// Mitsubishi GX Works2 project: Step Control   PLC: Q01U

PROGRAM conveyor
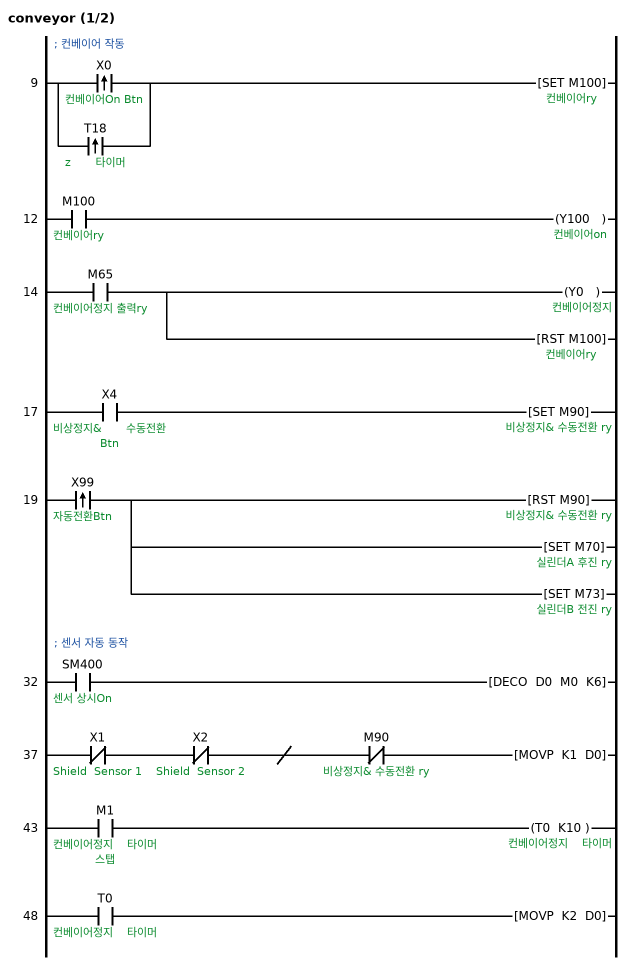
; 컨베이어 작동
9     LDP     X0  ; 컨베이어On Btn
      ORP     T18  ; z       타이머
      SET     M100  ; 컨베이어ry
12    LD      M100  ; 컨베이어ry
      OUT     Y100  ; 컨베이어on
14    LD      M65  ; 컨베이어정지 출력ry
      OUT     Y0  ; 컨베이어정지
      RST     M100  ; 컨베이어ry
17    LD      X4  ; 비상정지&       수동전환 Btn
      SET     M90  ; 비상정지& 수동전환 ry
19    LDP     X99  ; 자동전환Btn
      RST     M90  ; 비상정지& 수동전환 ry
      SET     M70  ; 실린더A 후진 ry
      SET     M73  ; 실린더B 전진 ry
; 센서 자동 동작
32    LD      SM400  ; 센서 상시On
      DECO    D0 M0 K6
37    LDI     X1  ; Shield  Sensor 1
      ANI     X2  ; Shield  Sensor 2
      INV
      ANI     M90  ; 비상정지& 수동전환 ry
      MOVP    K1 D0
43    LD      M1  ; 컨베이어정지    타이머  스탭
      OUT     T0 K10  ; 컨베이어정지    타이머
48    LD      T0  ; 컨베이어정지    타이머
      MOVP    K2 D0
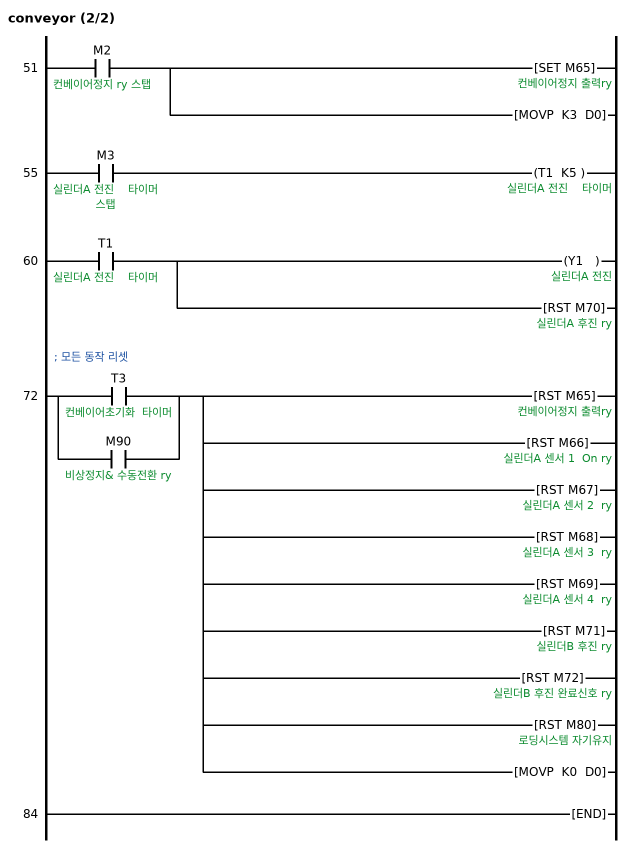
51    LD      M2  ; 컨베이어정지 ry 스탭
      SET     M65  ; 컨베이어정지 출력ry
      MOVP    K3 D0
55    LD      M3  ; 실린더A 전진    타이머  스탭
      OUT     T1 K5  ; 실린더A 전진    타이머
60    LD      T1  ; 실린더A 전진    타이머
      OUT     Y1  ; 실린더A 전진
      RST     M70  ; 실린더A 후진 ry
; 모든 동작 리셋
72    LD      T3  ; 컨베이어초기화  타이머
      OR      M90  ; 비상정지& 수동전환 ry
      RST     M65  ; 컨베이어정지 출력ry
      RST     M66  ; 실린더A 센서 1  On ry
      RST     M67  ; 실린더A 센서 2  ry
      RST     M68  ; 실린더A 센서 3  ry
      RST     M69  ; 실린더A 센서 4  ry
      RST     M71  ; 실린더B 후진 ry
      RST     M72  ; 실린더B 후진 완료신호 ry
      RST     M80  ; 로딩시스템 자기유지
      MOVP    K0 D0
84    END
END_PROGRAM

PROGRAM cylinder
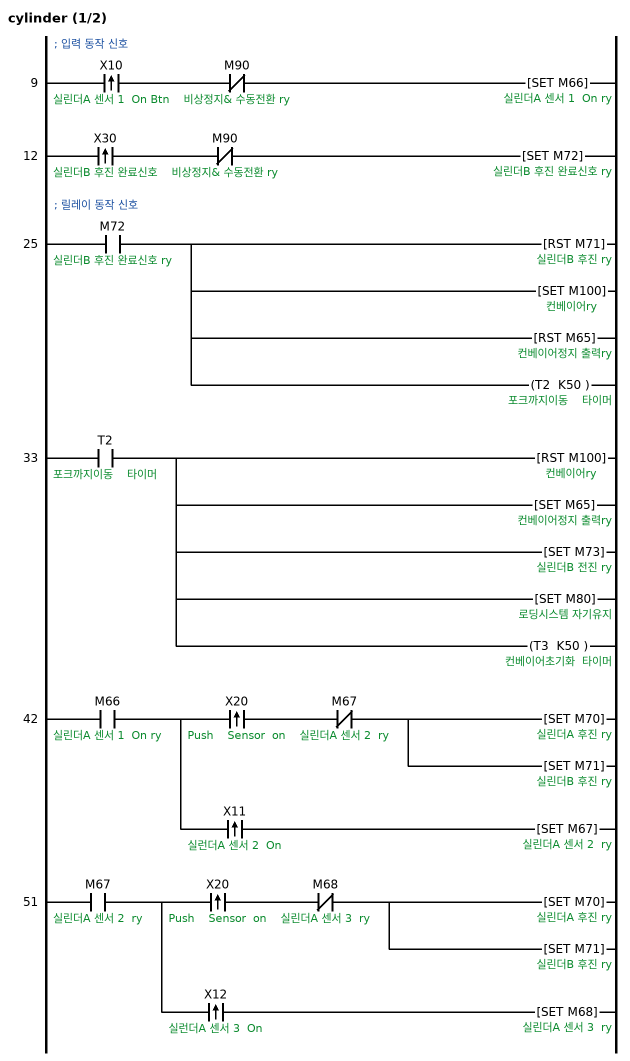
; 입력 동작 신호
9     LDP     X10  ; 실린더A 센서 1  On Btn
      ANI     M90  ; 비상정지& 수동전환 ry
      SET     M66  ; 실린더A 센서 1  On ry
12    LDP     X30  ; 실린더B 후진 완료신호
      ANI     M90  ; 비상정지& 수동전환 ry
      SET     M72  ; 실린더B 후진 완료신호 ry
; 릴레이 동작 신호
25    LD      M72  ; 실린더B 후진 완료신호 ry
      RST     M71  ; 실린더B 후진 ry
      SET     M100  ; 컨베이어ry
      RST     M65  ; 컨베이어정지 출력ry
      OUT     T2 K50  ; 포크까지이동    타이머
33    LD      T2  ; 포크까지이동    타이머
      RST     M100  ; 컨베이어ry
      SET     M65  ; 컨베이어정지 출력ry
      SET     M73  ; 실린더B 전진 ry
      SET     M80  ; 로딩시스템 자기유지
      OUT     T3 K50  ; 컨베이어초기화  타이머
42    LD      M66  ; 실린더A 센서 1  On ry
      MPS
      ANDP    X20  ; Push    Sensor  on
      ANI     M67  ; 실린더A 센서 2  ry
      SET     M70  ; 실린더A 후진 ry
      SET     M71  ; 실린더B 후진 ry
      MPP
      ANDP    X11  ; 실런더A 센서 2  On
      SET     M67  ; 실린더A 센서 2  ry
51    LD      M67  ; 실린더A 센서 2  ry
      MPS
      ANDP    X20  ; Push    Sensor  on
      ANI     M68  ; 실린더A 센서 3  ry
      SET     M70  ; 실린더A 후진 ry
      SET     M71  ; 실린더B 후진 ry
      MPP
      ANDP    X12  ; 실런더A 센서 3  On
      SET     M68  ; 실린더A 센서 3  ry
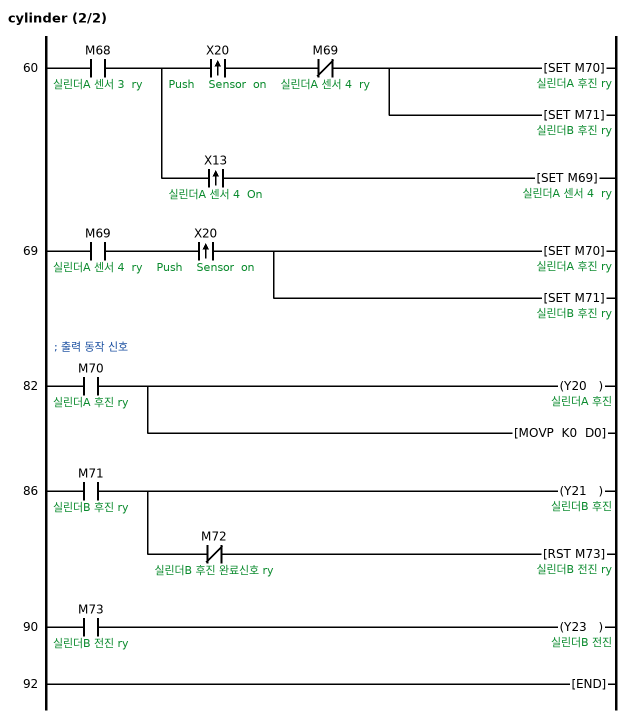
60    LD      M68  ; 실린더A 센서 3  ry
      MPS
      ANDP    X20  ; Push    Sensor  on
      ANI     M69  ; 실린더A 센서 4  ry
      SET     M70  ; 실린더A 후진 ry
      SET     M71  ; 실린더B 후진 ry
      MPP
      ANDP    X13  ; 실린더A 센서 4  On
      SET     M69  ; 실린더A 센서 4  ry
69    LD      M69  ; 실린더A 센서 4  ry
      ANDP    X20  ; Push    Sensor  on
      SET     M70  ; 실린더A 후진 ry
      SET     M71  ; 실린더B 후진 ry
; 출력 동작 신호
82    LD      M70  ; 실린더A 후진 ry
      OUT     Y20  ; 실린더A 후진
      MOVP    K0 D0
86    LD      M71  ; 실린더B 후진 ry
      OUT     Y21  ; 실린더B 후진
      ANI     M72  ; 실린더B 후진 완료신호 ry
      RST     M73  ; 실린더B 전진 ry
90    LD      M73  ; 실린더B 전진 ry
      OUT     Y23  ; 실린더B 전진
92    END
END_PROGRAM

PROGRAM manual
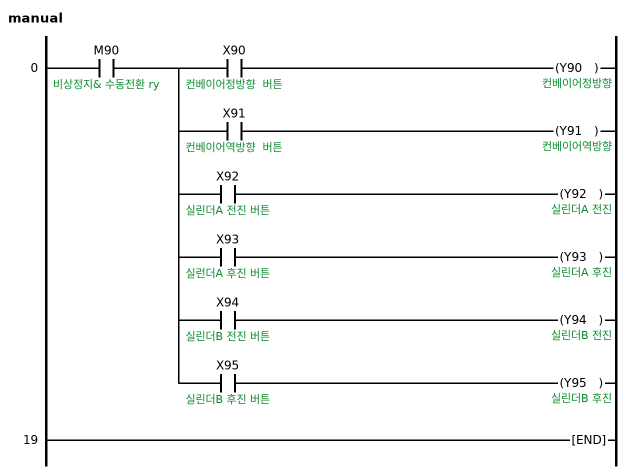
0     LD      M90  ; 비상정지& 수동전환 ry
      MPS
      AND     X90  ; 컨베이어정방향  버튼
      OUT     Y90  ; 컨베이어정방향
      MRD
      AND     X91  ; 컨베이어역방향  버튼
      OUT     Y91  ; 컨베이어역방향
      MRD
      AND     X92  ; 실린더A 전진 버튼
      OUT     Y92  ; 실린더A 전진
      MRD
      AND     X93  ; 실런더A 후진 버튼
      OUT     Y93  ; 실린더A 후진
      MRD
      AND     X94  ; 실린더B 전진 버튼
      OUT     Y94  ; 실린더B 전진
      MPP
      AND     X95  ; 실린더B 후진 버튼
      OUT     Y95  ; 실린더B 후진
19    END
END_PROGRAM

PROGRAM boxSize
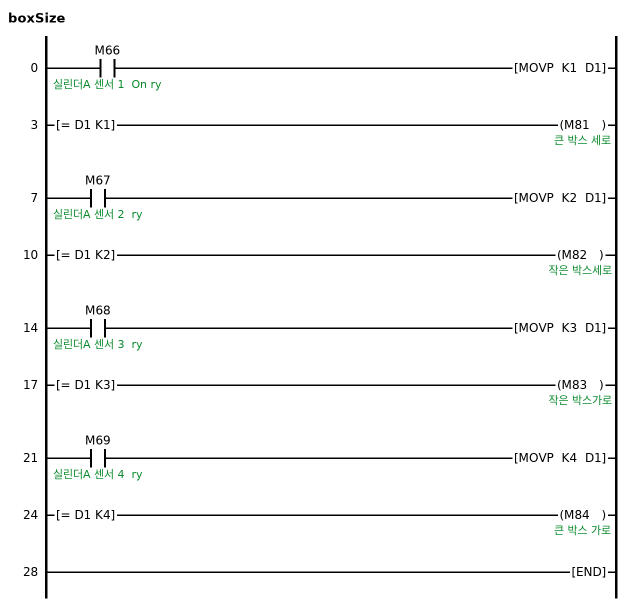
0     LD      M66  ; 실린더A 센서 1  On ry
      MOVP    K1 D1
3     LD=     D1 K1
      OUT     M81  ; 큰 박스 세로
7     LD      M67  ; 실린더A 센서 2  ry
      MOVP    K2 D1
10    LD=     D1 K2
      OUT     M82  ; 작은 박스세로
14    LD      M68  ; 실린더A 센서 3  ry
      MOVP    K3 D1
17    LD=     D1 K3
      OUT     M83  ; 작은 박스가로
21    LD      M69  ; 실린더A 센서 4  ry
      MOVP    K4 D1
24    LD=     D1 K4
      OUT     M84  ; 큰 박스 가로
28    END
END_PROGRAM

PROGRAM Box4move
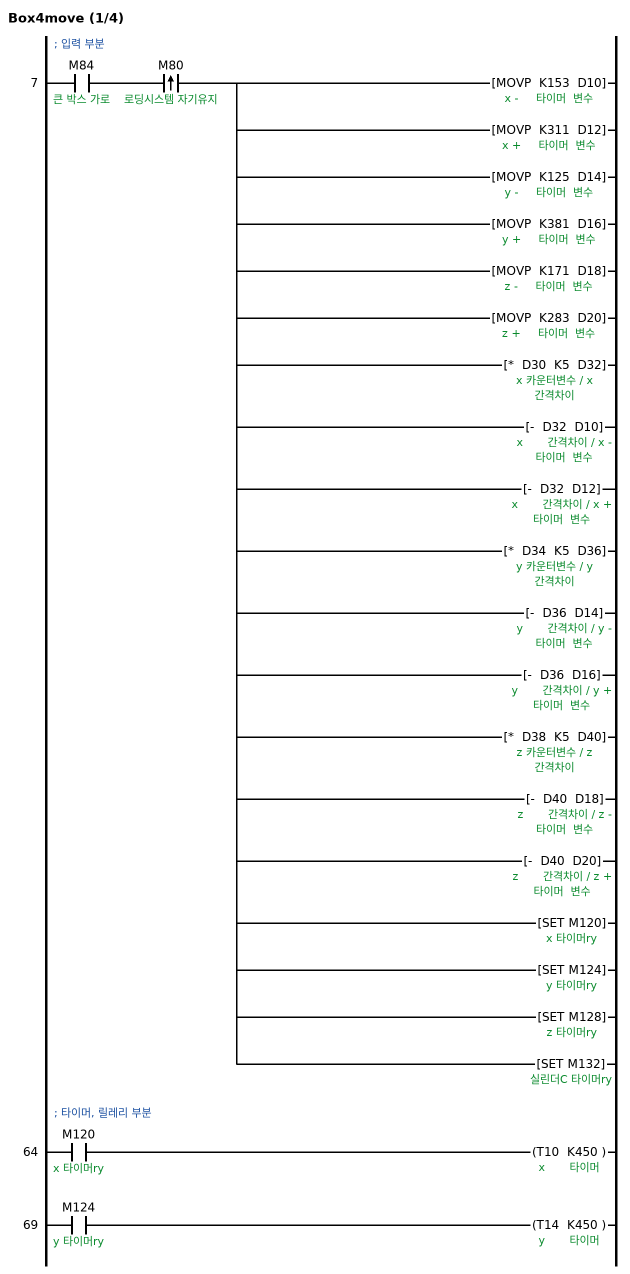
; 입력 부분
7     LD      M84  ; 큰 박스 가로
      ANDP    M80  ; 로딩시스템 자기유지
      MOVP    K153 D10  ; x -     타이머  변수
      MOVP    K311 D12  ; x +     타이머  변수
      MOVP    K125 D14  ; y -     타이머  변수
      MOVP    K381 D16  ; y +     타이머  변수
      MOVP    K171 D18  ; z -     타이머  변수
      MOVP    K283 D20  ; z +     타이머  변수
      *       D30 K5 D32  ; x 카운터변수 / x       간격차이
      -       D32 D10
      -       D32 D12
      *       D34 K5 D36  ; y 카운터변수 / y       간격차이
      -       D36 D14
      -       D36 D16
      *       D38 K5 D40  ; z 카운터변수 / z       간격차이
      -       D40 D18
      -       D40 D20
      SET     M120  ; x 타이머ry
      SET     M124  ; y 타이머ry
      SET     M128  ; z 타이머ry
      SET     M132  ; 실린더C 타이머ry
; 타이머, 릴레리 부분
64    LD      M120  ; x 타이머ry
      OUT     T10 K450  ; x       타이머
69    LD      M124  ; y 타이머ry
      OUT     T14 K450  ; y       타이머
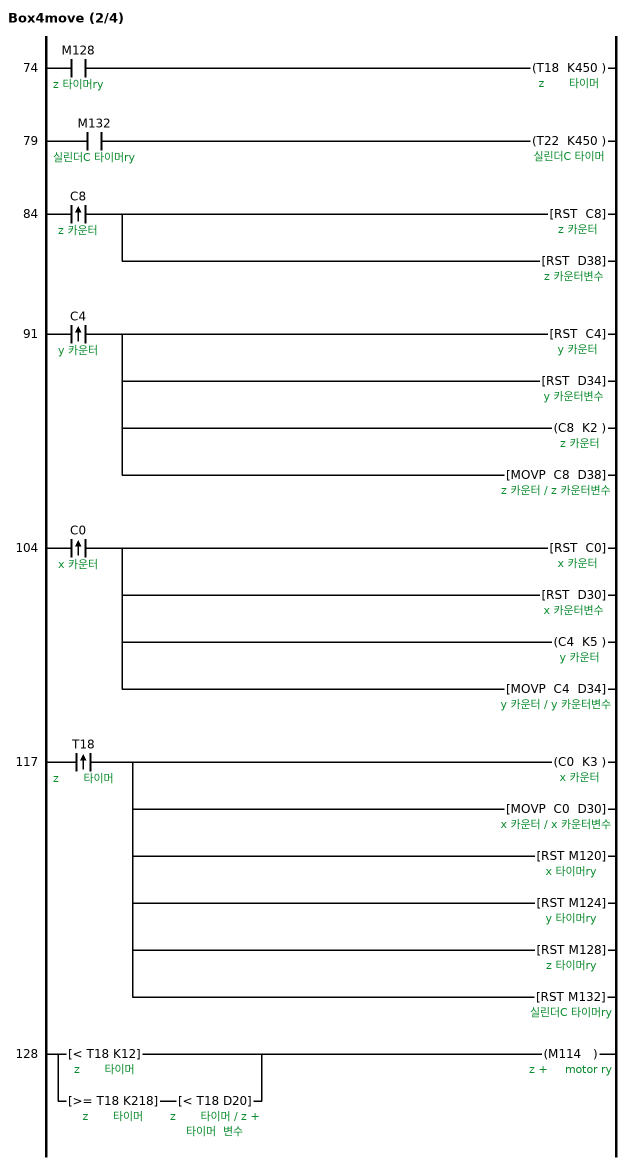
74    LD      M128  ; z 타이머ry
      OUT     T18 K450  ; z       타이머
79    LD      M132  ; 실린더C 타이머ry
      OUT     T22 K450  ; 실린더C 타이머
84    LDP     C8  ; z 카운터
      RST     C8  ; z 카운터
      RST     D38  ; z 카운터변수
91    LDP     C4  ; y 카운터
      RST     C4  ; y 카운터
      RST     D34  ; y 카운터변수
      OUT     C8 K2  ; z 카운터
      MOVP    C8 D38
104   LDP     C0  ; x 카운터
      RST     C0  ; x 카운터
      RST     D30  ; x 카운터변수
      OUT     C4 K5  ; y 카운터
      MOVP    C4 D34
117   LDP     T18  ; z       타이머
      OUT     C0 K3  ; x 카운터
      MOVP    C0 D30
      RST     M120  ; x 타이머ry
      RST     M124  ; y 타이머ry
      RST     M128  ; z 타이머ry
      RST     M132  ; 실린더C 타이머ry
128   LD<     T18 K12  ; z       타이머
      LD>=    T18 K218  ; z       타이머
      AND<    T18 D20  ; z       타이머 / z +     타이머  변수
      ORB
      OUT     M114  ; z +     motor ry
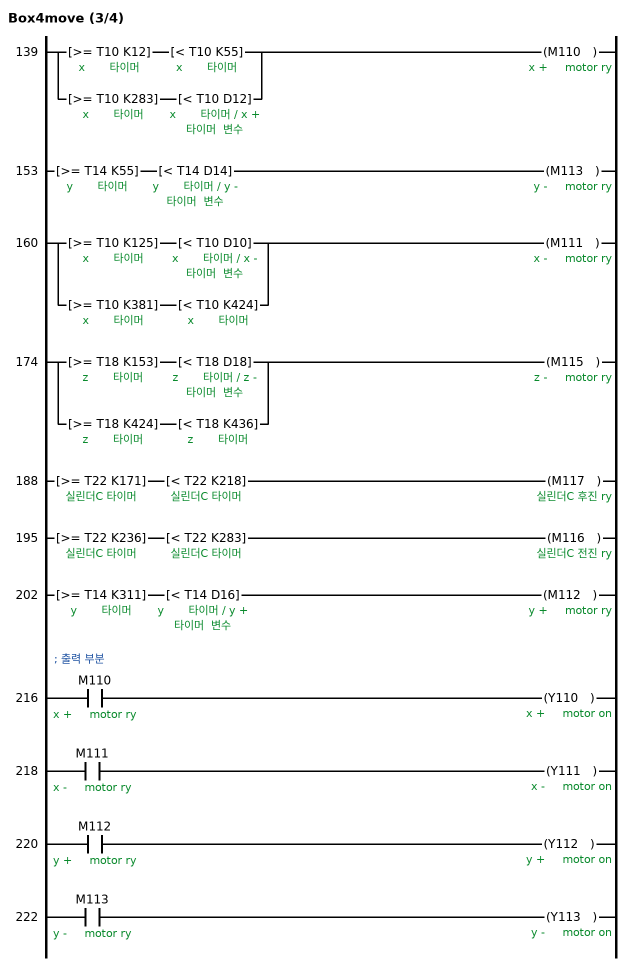
139   LD>=    T10 K12  ; x       타이머
      AND<    T10 K55  ; x       타이머
      LD>=    T10 K283  ; x       타이머
      AND<    T10 D12  ; x       타이머 / x +     타이머  변수
      ORB
      OUT     M110  ; x +     motor ry
153   LD>=    T14 K55  ; y       타이머
      AND<    T14 D14  ; y       타이머 / y -     타이머  변수
      OUT     M113  ; y -     motor ry
160   LD>=    T10 K125  ; x       타이머
      AND<    T10 D10  ; x       타이머 / x -     타이머  변수
      LD>=    T10 K381  ; x       타이머
      AND<    T10 K424  ; x       타이머
      ORB
      OUT     M111  ; x -     motor ry
174   LD>=    T18 K153  ; z       타이머
      AND<    T18 D18  ; z       타이머 / z -     타이머  변수
      LD>=    T18 K424  ; z       타이머
      AND<    T18 K436  ; z       타이머
      ORB
      OUT     M115  ; z -     motor ry
188   LD>=    T22 K171  ; 실린더C 타이머
      AND<    T22 K218  ; 실린더C 타이머
      OUT     M117  ; 실린더C 후진 ry
195   LD>=    T22 K236  ; 실린더C 타이머
      AND<    T22 K283  ; 실린더C 타이머
      OUT     M116  ; 실린더C 전진 ry
202   LD>=    T14 K311  ; y       타이머
      AND<    T14 D16  ; y       타이머 / y +     타이머  변수
      OUT     M112  ; y +     motor ry
; 출력 부분
216   LD      M110  ; x +     motor ry
      OUT     Y110  ; x +     motor on
218   LD      M111  ; x -     motor ry
      OUT     Y111  ; x -     motor on
220   LD      M112  ; y +     motor ry
      OUT     Y112  ; y +     motor on
222   LD      M113  ; y -     motor ry
      OUT     Y113  ; y -     motor on
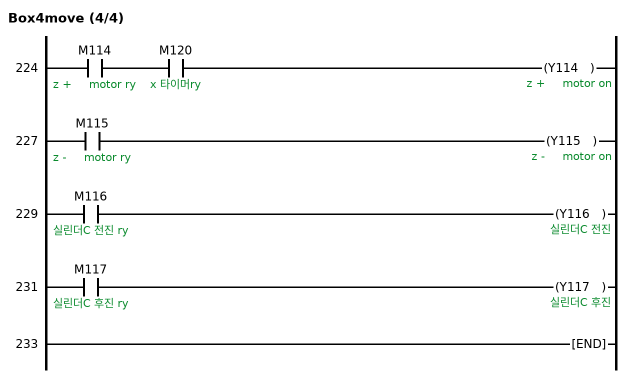
224   LD      M114  ; z +     motor ry
      AND     M120  ; x 타이머ry
      OUT     Y114  ; z +     motor on
227   LD      M115  ; z -     motor ry
      OUT     Y115  ; z -     motor on
229   LD      M116  ; 실린더C 전진 ry
      OUT     Y116  ; 실린더C 전진
231   LD      M117  ; 실린더C 후진 ry
      OUT     Y117  ; 실린더C 후진
233   END
END_PROGRAM

PROGRAM Lmanual
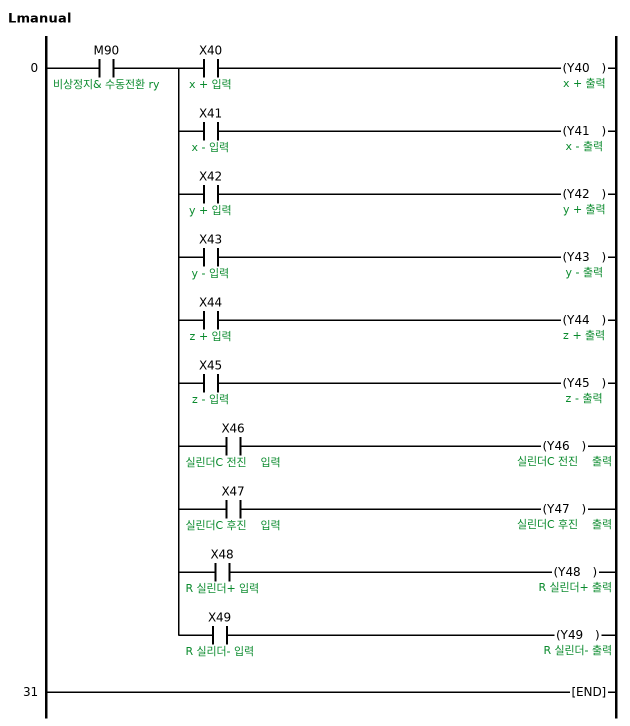
0     LD      M90  ; 비상정지& 수동전환 ry
      MPS
      AND     X40  ; x + 입력
      OUT     Y40  ; x + 출력
      MRD
      AND     X41  ; x - 입력
      OUT     Y41  ; x - 출력
      MRD
      AND     X42  ; y + 입력
      OUT     Y42  ; y + 출력
      MRD
      AND     X43  ; y - 입력
      OUT     Y43  ; y - 출력
      MRD
      AND     X44  ; z + 입력
      OUT     Y44  ; z + 출력
      MRD
      AND     X45  ; z - 입력
      OUT     Y45  ; z - 출력
      MRD
      AND     X46  ; 실린더C 전진    입력
      OUT     Y46  ; 실린더C 전진    출력
      MRD
      AND     X47  ; 실린더C 후진    입력
      OUT     Y47  ; 실린더C 후진    출력
      MRD
      AND     X48  ; R 실린더+ 입력
      OUT     Y48  ; R 실린더+ 출력
      MPP
      AND     X49  ; R 실리더- 입력
      OUT     Y49  ; R 실린더- 출력
31    END
END_PROGRAM

PROGRAM Box1move
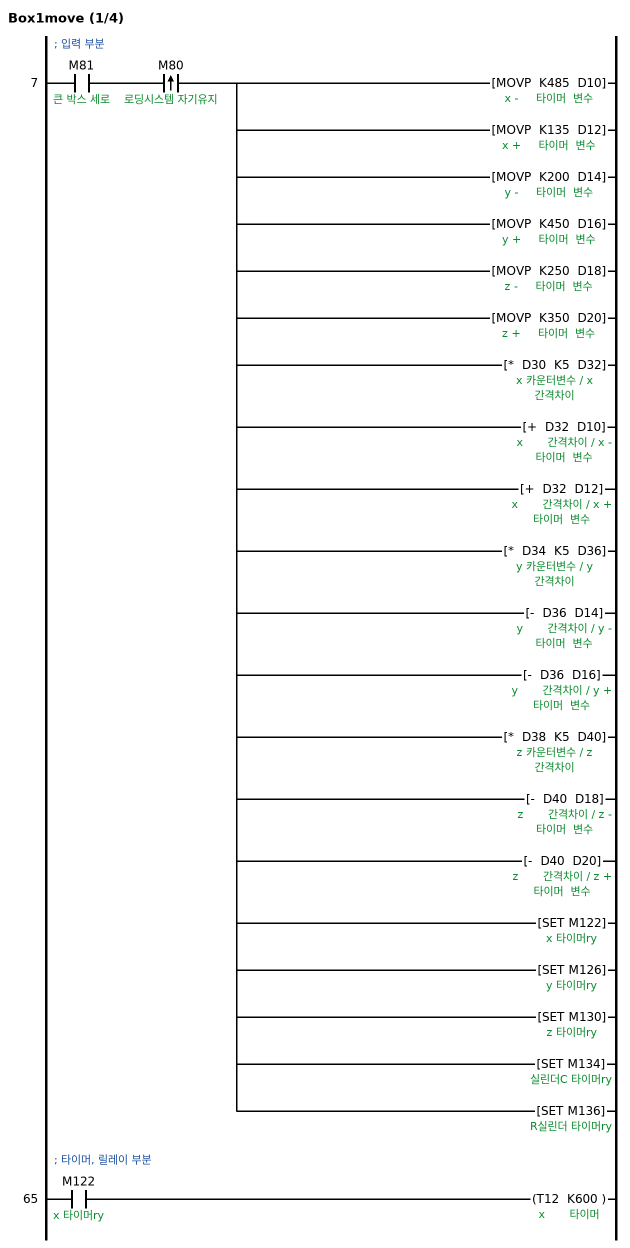
; 입력 부분
7     LD      M81  ; 큰 박스 세로
      ANDP    M80  ; 로딩시스템 자기유지
      MOVP    K485 D10  ; x -     타이머  변수
      MOVP    K135 D12  ; x +     타이머  변수
      MOVP    K200 D14  ; y -     타이머  변수
      MOVP    K450 D16  ; y +     타이머  변수
      MOVP    K250 D18  ; z -     타이머  변수
      MOVP    K350 D20  ; z +     타이머  변수
      *       D30 K5 D32  ; x 카운터변수 / x       간격차이
      +       D32 D10
      +       D32 D12
      *       D34 K5 D36  ; y 카운터변수 / y       간격차이
      -       D36 D14
      -       D36 D16
      *       D38 K5 D40  ; z 카운터변수 / z       간격차이
      -       D40 D18
      -       D40 D20
      SET     M122  ; x 타이머ry
      SET     M126  ; y 타이머ry
      SET     M130  ; z 타이머ry
      SET     M134  ; 실린더C 타이머ry
      SET     M136  ; R실린더 타이머ry
; 타이머, 릴레이 부분
65    LD      M122  ; x 타이머ry
      OUT     T12 K600  ; x       타이머
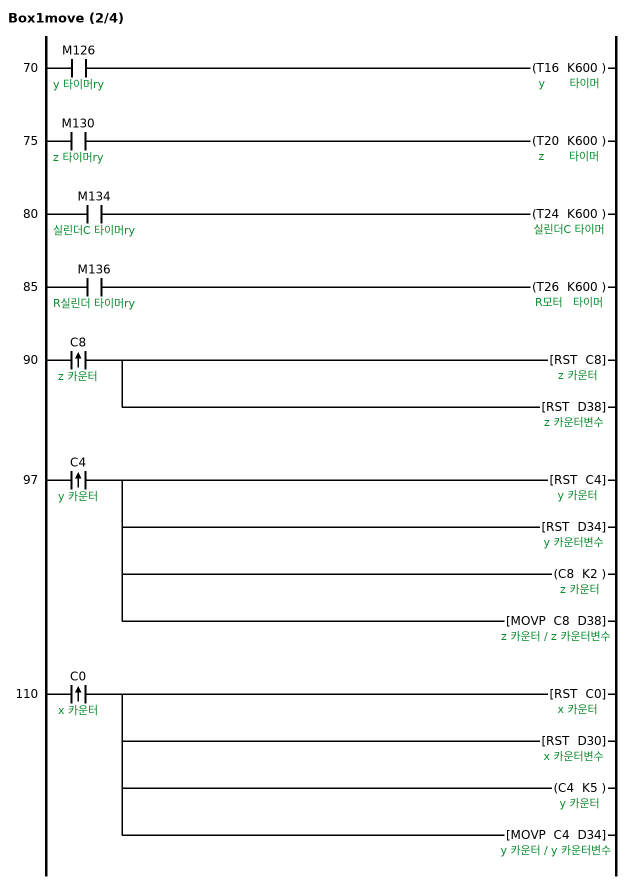
70    LD      M126  ; y 타이머ry
      OUT     T16 K600  ; y       타이머
75    LD      M130  ; z 타이머ry
      OUT     T20 K600  ; z       타이머
80    LD      M134  ; 실린더C 타이머ry
      OUT     T24 K600  ; 실린더C 타이머
85    LD      M136  ; R실린더 타이머ry
      OUT     T26 K600  ; R모터   타이머
90    LDP     C8  ; z 카운터
      RST     C8  ; z 카운터
      RST     D38  ; z 카운터변수
97    LDP     C4  ; y 카운터
      RST     C4  ; y 카운터
      RST     D34  ; y 카운터변수
      OUT     C8 K2  ; z 카운터
      MOVP    C8 D38
110   LDP     C0  ; x 카운터
      RST     C0  ; x 카운터
      RST     D30  ; x 카운터변수
      OUT     C4 K5  ; y 카운터
      MOVP    C4 D34
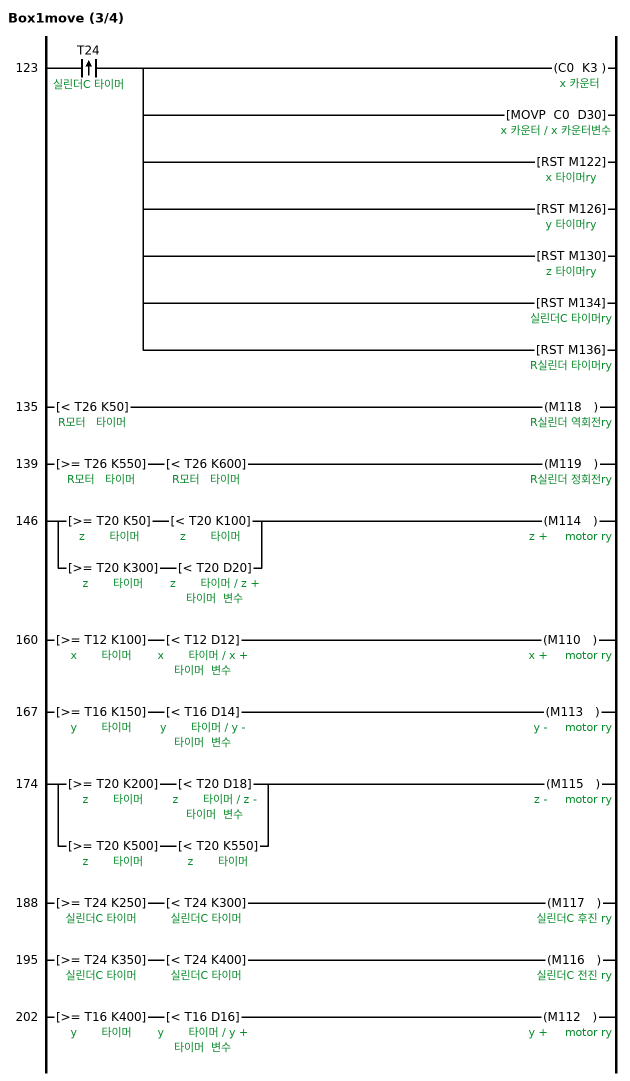
123   LDP     T24  ; 실린더C 타이머
      OUT     C0 K3  ; x 카운터
      MOVP    C0 D30
      RST     M122  ; x 타이머ry
      RST     M126  ; y 타이머ry
      RST     M130  ; z 타이머ry
      RST     M134  ; 실린더C 타이머ry
      RST     M136  ; R실린더 타이머ry
135   LD<     T26 K50  ; R모터   타이머
      OUT     M118  ; R실린더 역회전ry
139   LD>=    T26 K550  ; R모터   타이머
      AND<    T26 K600  ; R모터   타이머
      OUT     M119  ; R실린더 정회전ry
146   LD>=    T20 K50  ; z       타이머
      AND<    T20 K100  ; z       타이머
      LD>=    T20 K300  ; z       타이머
      AND<    T20 D20  ; z       타이머 / z +     타이머  변수
      ORB
      OUT     M114  ; z +     motor ry
160   LD>=    T12 K100  ; x       타이머
      AND<    T12 D12  ; x       타이머 / x +     타이머  변수
      OUT     M110  ; x +     motor ry
167   LD>=    T16 K150  ; y       타이머
      AND<    T16 D14  ; y       타이머 / y -     타이머  변수
      OUT     M113  ; y -     motor ry
174   LD>=    T20 K200  ; z       타이머
      AND<    T20 D18  ; z       타이머 / z -     타이머  변수
      LD>=    T20 K500  ; z       타이머
      AND<    T20 K550  ; z       타이머
      ORB
      OUT     M115  ; z -     motor ry
188   LD>=    T24 K250  ; 실린더C 타이머
      AND<    T24 K300  ; 실린더C 타이머
      OUT     M117  ; 실린더C 후진 ry
195   LD>=    T24 K350  ; 실린더C 타이머
      AND<    T24 K400  ; 실린더C 타이머
      OUT     M116  ; 실린더C 전진 ry
202   LD>=    T16 K400  ; y       타이머
      AND<    T16 D16  ; y       타이머 / y +     타이머  변수
      OUT     M112  ; y +     motor ry
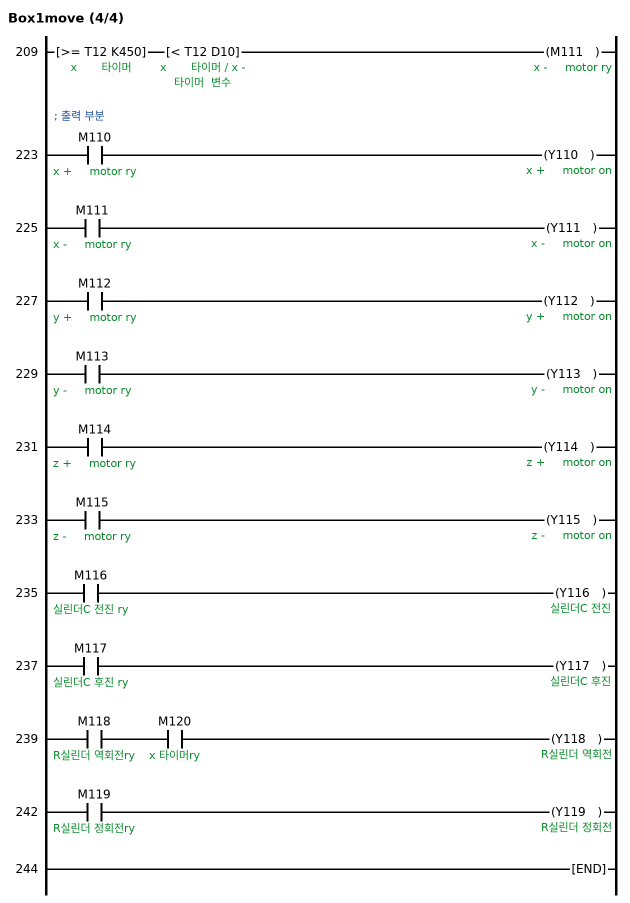
209   LD>=    T12 K450  ; x       타이머
      AND<    T12 D10  ; x       타이머 / x -     타이머  변수
      OUT     M111  ; x -     motor ry
; 출력 부분
223   LD      M110  ; x +     motor ry
      OUT     Y110  ; x +     motor on
225   LD      M111  ; x -     motor ry
      OUT     Y111  ; x -     motor on
227   LD      M112  ; y +     motor ry
      OUT     Y112  ; y +     motor on
229   LD      M113  ; y -     motor ry
      OUT     Y113  ; y -     motor on
231   LD      M114  ; z +     motor ry
      OUT     Y114  ; z +     motor on
233   LD      M115  ; z -     motor ry
      OUT     Y115  ; z -     motor on
235   LD      M116  ; 실린더C 전진 ry
      OUT     Y116  ; 실린더C 전진
237   LD      M117  ; 실린더C 후진 ry
      OUT     Y117  ; 실린더C 후진
239   LD      M118  ; R실린더 역회전ry
      AND     M120  ; x 타이머ry
      OUT     Y118  ; R실린더 역회전
242   LD      M119  ; R실린더 정회전ry
      OUT     Y119  ; R실린더 정회전
244   END
END_PROGRAM

PROGRAM Box2move
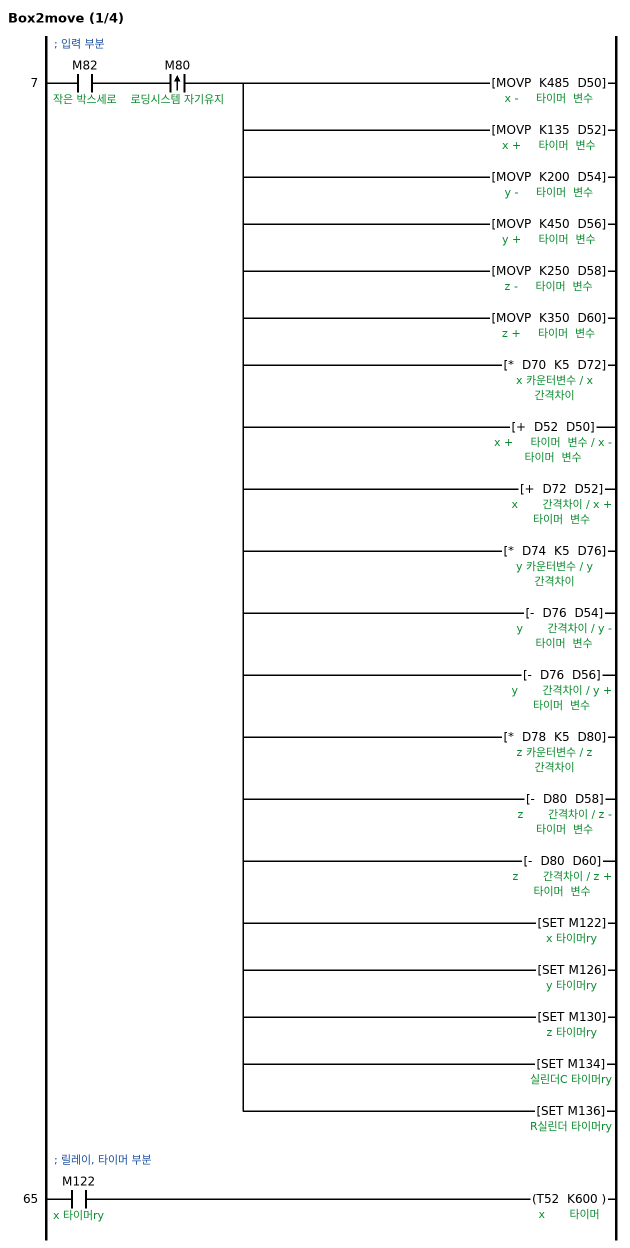
; 입력 부분
7     LD      M82  ; 작은 박스세로
      ANDP    M80  ; 로딩시스템 자기유지
      MOVP    K485 D50  ; x -     타이머  변수
      MOVP    K135 D52  ; x +     타이머  변수
      MOVP    K200 D54  ; y -     타이머  변수
      MOVP    K450 D56  ; y +     타이머  변수
      MOVP    K250 D58  ; z -     타이머  변수
      MOVP    K350 D60  ; z +     타이머  변수
      *       D70 K5 D72  ; x 카운터변수 / x       간격차이
      +       D52 D50
      +       D72 D52
      *       D74 K5 D76  ; y 카운터변수 / y       간격차이
      -       D76 D54
      -       D76 D56
      *       D78 K5 D80  ; z 카운터변수 / z       간격차이
      -       D80 D58
      -       D80 D60
      SET     M122  ; x 타이머ry
      SET     M126  ; y 타이머ry
      SET     M130  ; z 타이머ry
      SET     M134  ; 실린더C 타이머ry
      SET     M136  ; R실린더 타이머ry
; 릴레이, 타이머 부분
65    LD      M122  ; x 타이머ry
      OUT     T52 K600  ; x       타이머
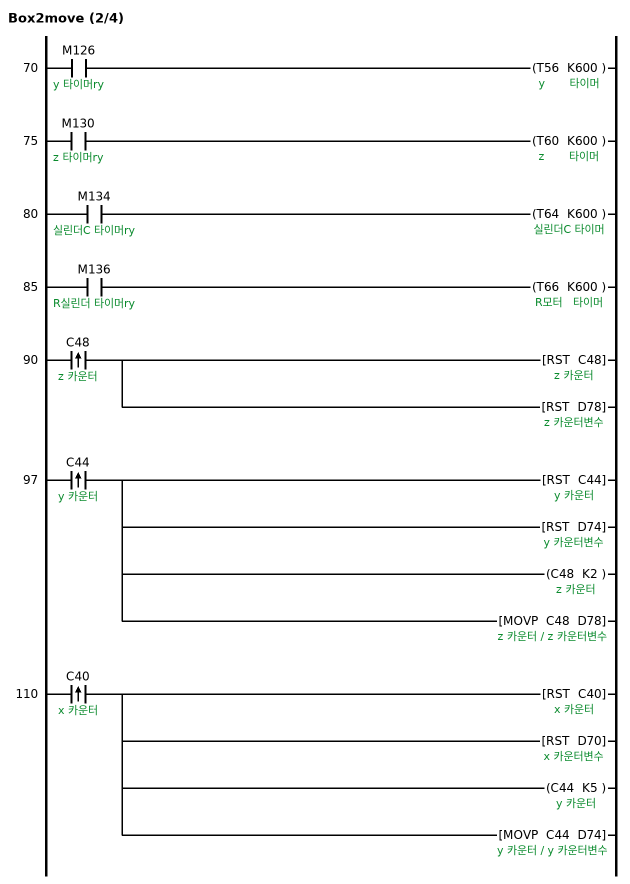
70    LD      M126  ; y 타이머ry
      OUT     T56 K600  ; y       타이머
75    LD      M130  ; z 타이머ry
      OUT     T60 K600  ; z       타이머
80    LD      M134  ; 실린더C 타이머ry
      OUT     T64 K600  ; 실린더C 타이머
85    LD      M136  ; R실린더 타이머ry
      OUT     T66 K600  ; R모터   타이머
90    LDP     C48  ; z 카운터
      RST     C48  ; z 카운터
      RST     D78  ; z 카운터변수
97    LDP     C44  ; y 카운터
      RST     C44  ; y 카운터
      RST     D74  ; y 카운터변수
      OUT     C48 K2  ; z 카운터
      MOVP    C48 D78
110   LDP     C40  ; x 카운터
      RST     C40  ; x 카운터
      RST     D70  ; x 카운터변수
      OUT     C44 K5  ; y 카운터
      MOVP    C44 D74
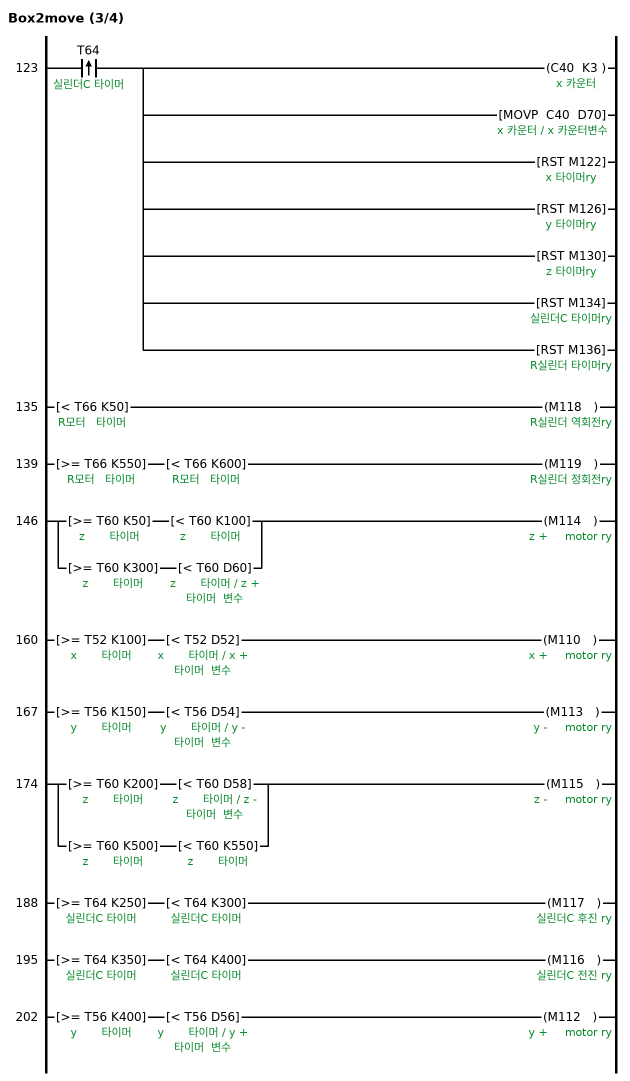
123   LDP     T64  ; 실린더C 타이머
      OUT     C40 K3  ; x 카운터
      MOVP    C40 D70
      RST     M122  ; x 타이머ry
      RST     M126  ; y 타이머ry
      RST     M130  ; z 타이머ry
      RST     M134  ; 실린더C 타이머ry
      RST     M136  ; R실린더 타이머ry
135   LD<     T66 K50  ; R모터   타이머
      OUT     M118  ; R실린더 역회전ry
139   LD>=    T66 K550  ; R모터   타이머
      AND<    T66 K600  ; R모터   타이머
      OUT     M119  ; R실린더 정회전ry
146   LD>=    T60 K50  ; z       타이머
      AND<    T60 K100  ; z       타이머
      LD>=    T60 K300  ; z       타이머
      AND<    T60 D60  ; z       타이머 / z +     타이머  변수
      ORB
      OUT     M114  ; z +     motor ry
160   LD>=    T52 K100  ; x       타이머
      AND<    T52 D52  ; x       타이머 / x +     타이머  변수
      OUT     M110  ; x +     motor ry
167   LD>=    T56 K150  ; y       타이머
      AND<    T56 D54  ; y       타이머 / y -     타이머  변수
      OUT     M113  ; y -     motor ry
174   LD>=    T60 K200  ; z       타이머
      AND<    T60 D58  ; z       타이머 / z -     타이머  변수
      LD>=    T60 K500  ; z       타이머
      AND<    T60 K550  ; z       타이머
      ORB
      OUT     M115  ; z -     motor ry
188   LD>=    T64 K250  ; 실린더C 타이머
      AND<    T64 K300  ; 실린더C 타이머
      OUT     M117  ; 실린더C 후진 ry
195   LD>=    T64 K350  ; 실린더C 타이머
      AND<    T64 K400  ; 실린더C 타이머
      OUT     M116  ; 실린더C 전진 ry
202   LD>=    T56 K400  ; y       타이머
      AND<    T56 D56  ; y       타이머 / y +     타이머  변수
      OUT     M112  ; y +     motor ry
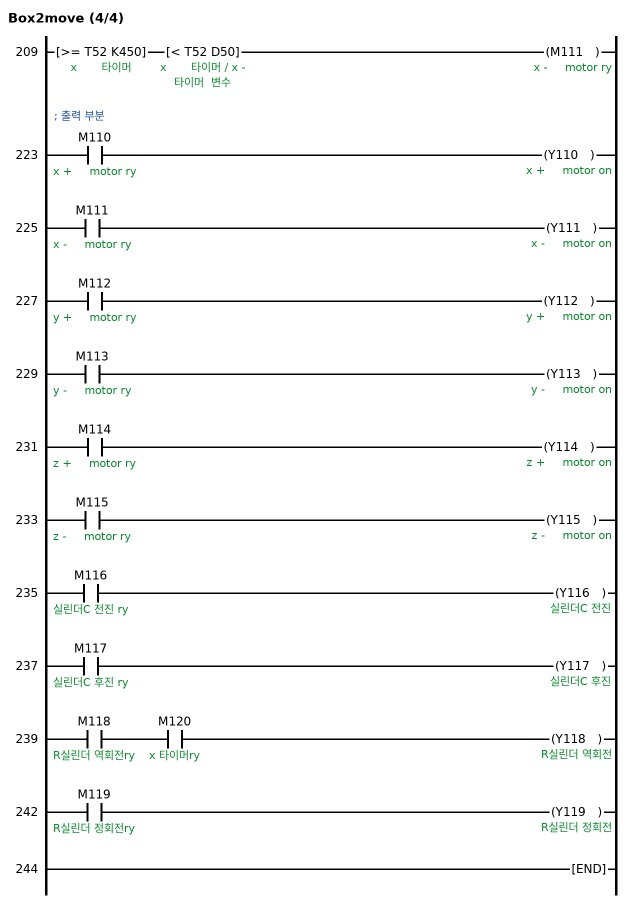
209   LD>=    T52 K450  ; x       타이머
      AND<    T52 D50  ; x       타이머 / x -     타이머  변수
      OUT     M111  ; x -     motor ry
; 출력 부분
223   LD      M110  ; x +     motor ry
      OUT     Y110  ; x +     motor on
225   LD      M111  ; x -     motor ry
      OUT     Y111  ; x -     motor on
227   LD      M112  ; y +     motor ry
      OUT     Y112  ; y +     motor on
229   LD      M113  ; y -     motor ry
      OUT     Y113  ; y -     motor on
231   LD      M114  ; z +     motor ry
      OUT     Y114  ; z +     motor on
233   LD      M115  ; z -     motor ry
      OUT     Y115  ; z -     motor on
235   LD      M116  ; 실린더C 전진 ry
      OUT     Y116  ; 실린더C 전진
237   LD      M117  ; 실린더C 후진 ry
      OUT     Y117  ; 실린더C 후진
239   LD      M118  ; R실린더 역회전ry
      AND     M120  ; x 타이머ry
      OUT     Y118  ; R실린더 역회전
242   LD      M119  ; R실린더 정회전ry
      OUT     Y119  ; R실린더 정회전
244   END
END_PROGRAM

PROGRAM Box3move
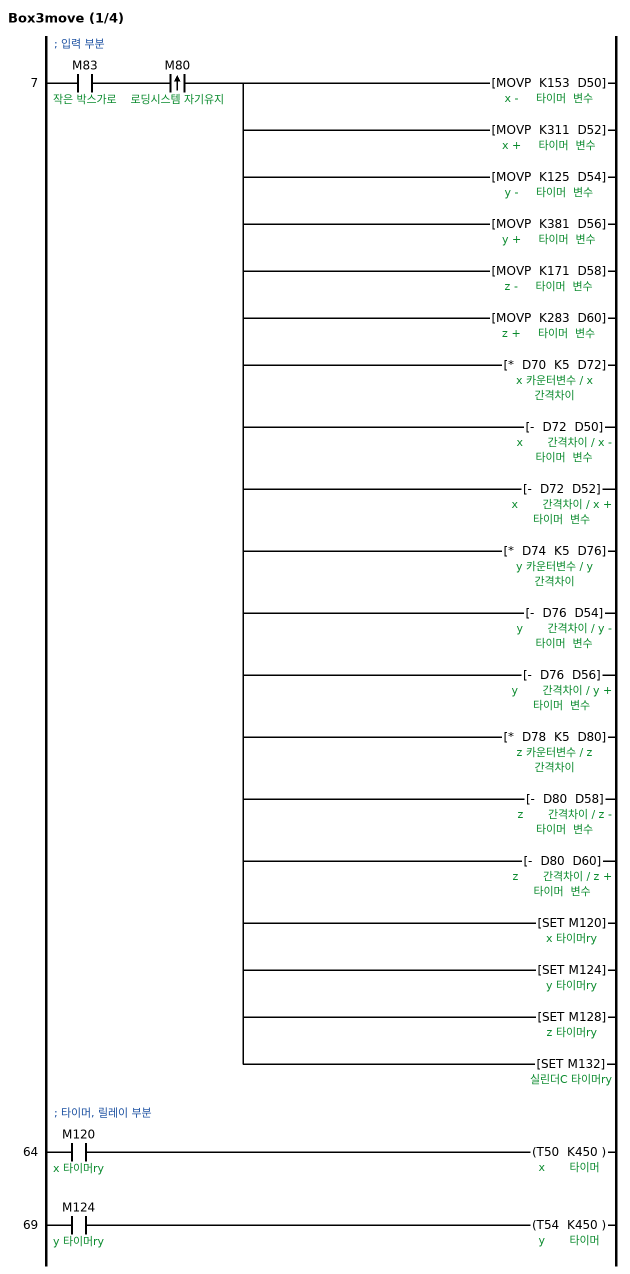
; 입력 부분
7     LD      M83  ; 작은 박스가로
      ANDP    M80  ; 로딩시스템 자기유지
      MOVP    K153 D50  ; x -     타이머  변수
      MOVP    K311 D52  ; x +     타이머  변수
      MOVP    K125 D54  ; y -     타이머  변수
      MOVP    K381 D56  ; y +     타이머  변수
      MOVP    K171 D58  ; z -     타이머  변수
      MOVP    K283 D60  ; z +     타이머  변수
      *       D70 K5 D72  ; x 카운터변수 / x       간격차이
      -       D72 D50
      -       D72 D52
      *       D74 K5 D76  ; y 카운터변수 / y       간격차이
      -       D76 D54
      -       D76 D56
      *       D78 K5 D80  ; z 카운터변수 / z       간격차이
      -       D80 D58
      -       D80 D60
      SET     M120  ; x 타이머ry
      SET     M124  ; y 타이머ry
      SET     M128  ; z 타이머ry
      SET     M132  ; 실린더C 타이머ry
; 타이머, 릴레이 부분
64    LD      M120  ; x 타이머ry
      OUT     T50 K450  ; x       타이머
69    LD      M124  ; y 타이머ry
      OUT     T54 K450  ; y       타이머
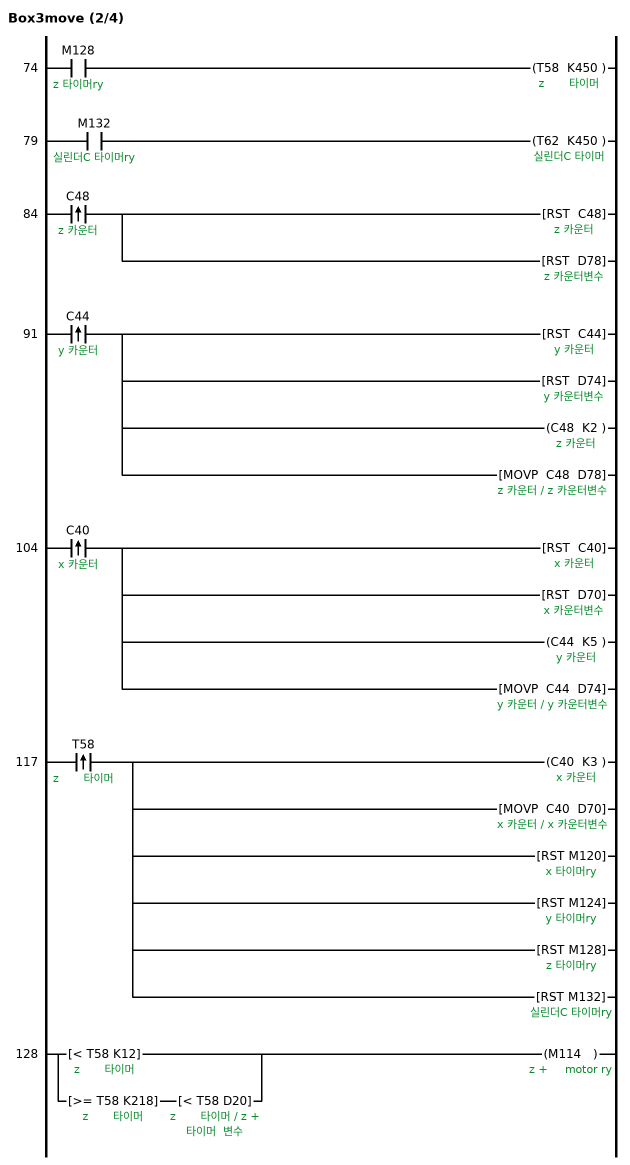
74    LD      M128  ; z 타이머ry
      OUT     T58 K450  ; z       타이머
79    LD      M132  ; 실린더C 타이머ry
      OUT     T62 K450  ; 실린더C 타이머
84    LDP     C48  ; z 카운터
      RST     C48  ; z 카운터
      RST     D78  ; z 카운터변수
91    LDP     C44  ; y 카운터
      RST     C44  ; y 카운터
      RST     D74  ; y 카운터변수
      OUT     C48 K2  ; z 카운터
      MOVP    C48 D78
104   LDP     C40  ; x 카운터
      RST     C40  ; x 카운터
      RST     D70  ; x 카운터변수
      OUT     C44 K5  ; y 카운터
      MOVP    C44 D74
117   LDP     T58  ; z       타이머
      OUT     C40 K3  ; x 카운터
      MOVP    C40 D70
      RST     M120  ; x 타이머ry
      RST     M124  ; y 타이머ry
      RST     M128  ; z 타이머ry
      RST     M132  ; 실린더C 타이머ry
128   LD<     T58 K12  ; z       타이머
      LD>=    T58 K218  ; z       타이머
      AND<    T58 D20  ; z       타이머 / z +     타이머  변수
      ORB
      OUT     M114  ; z +     motor ry
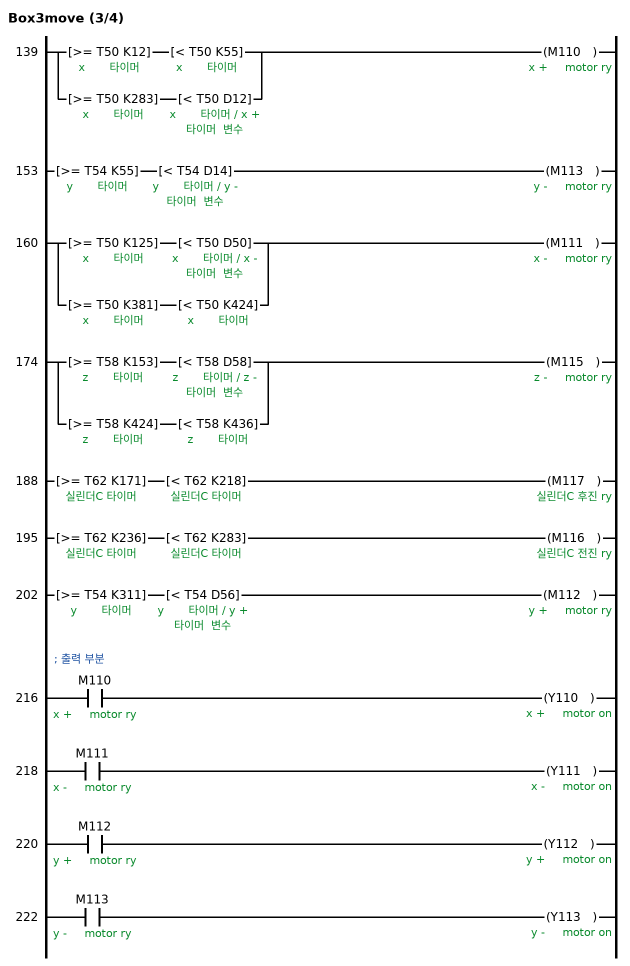
139   LD>=    T50 K12  ; x       타이머
      AND<    T50 K55  ; x       타이머
      LD>=    T50 K283  ; x       타이머
      AND<    T50 D12  ; x       타이머 / x +     타이머  변수
      ORB
      OUT     M110  ; x +     motor ry
153   LD>=    T54 K55  ; y       타이머
      AND<    T54 D14  ; y       타이머 / y -     타이머  변수
      OUT     M113  ; y -     motor ry
160   LD>=    T50 K125  ; x       타이머
      AND<    T50 D50  ; x       타이머 / x -     타이머  변수
      LD>=    T50 K381  ; x       타이머
      AND<    T50 K424  ; x       타이머
      ORB
      OUT     M111  ; x -     motor ry
174   LD>=    T58 K153  ; z       타이머
      AND<    T58 D58  ; z       타이머 / z -     타이머  변수
      LD>=    T58 K424  ; z       타이머
      AND<    T58 K436  ; z       타이머
      ORB
      OUT     M115  ; z -     motor ry
188   LD>=    T62 K171  ; 실린더C 타이머
      AND<    T62 K218  ; 실린더C 타이머
      OUT     M117  ; 실린더C 후진 ry
195   LD>=    T62 K236  ; 실린더C 타이머
      AND<    T62 K283  ; 실린더C 타이머
      OUT     M116  ; 실린더C 전진 ry
202   LD>=    T54 K311  ; y       타이머
      AND<    T54 D56  ; y       타이머 / y +     타이머  변수
      OUT     M112  ; y +     motor ry
; 출력 부분
216   LD      M110  ; x +     motor ry
      OUT     Y110  ; x +     motor on
218   LD      M111  ; x -     motor ry
      OUT     Y111  ; x -     motor on
220   LD      M112  ; y +     motor ry
      OUT     Y112  ; y +     motor on
222   LD      M113  ; y -     motor ry
      OUT     Y113  ; y -     motor on
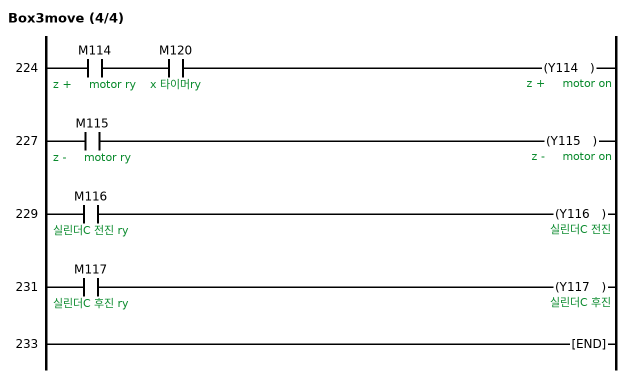
224   LD      M114  ; z +     motor ry
      AND     M120  ; x 타이머ry
      OUT     Y114  ; z +     motor on
227   LD      M115  ; z -     motor ry
      OUT     Y115  ; z -     motor on
229   LD      M116  ; 실린더C 전진 ry
      OUT     Y116  ; 실린더C 전진
231   LD      M117  ; 실린더C 후진 ry
      OUT     Y117  ; 실린더C 후진
233   END
END_PROGRAM

// device comments not shown above
T4  ; 실린더C 전진    타이머
T5  ; 실린더C 후진    타이머
D22  ; 실린더C 타이머  변수
D24  ; z -     타이머  변수
D62  ; 실린더C 타이머  변수
D64  ; z -     타이머  변수
